(* IEC 61131-3 sources: SIGMATEK-Jumag-Utils-Examples/edgeDetection/Class/Class0, 1 file *)

(* ---- Class0.st ---- *)
(*!
<Class
	Name               = "Class0"
	Revision           = "0.0"
	RealtimeTask       = "false"
	CyclicTask         = "true"
	DefCyclictime      = "100 ms"
	BackgroundTask     = "false"
	Sigmatek           = "false"
	OSInterface        = "false"
	HighPriority       = "false"
	Automatic          = "false"
	UpdateMode         = "Prescan"
	SharedCommandTable = "true"
	Objectsize         = "(660,120)">
	<Channels>
		<Server Name="ClassSvr" Visualized="false" Initialize="false" WriteProtected="true" Retentive="false"/>
		<Server Name="fallingTriggered" Visualized="false" Initialize="false" WriteProtected="false" Retentive="false"/>
		<Server Name="risingTriggered" Visualized="false" Initialize="false" WriteProtected="false" Retentive="false"/>
		<Server Name="targetValue" Visualized="false" Initialize="true" WriteProtected="false" Retentive="false"/>
		<Client Name="signal" Required="true" Internal="false"/>
	</Channels>
	<Dependencies>
		<Files>
			<File Path=".\Source\edgeDetection.c"/>
		</Files>
	</Dependencies>
</Class>
*)
Class0 : CLASS
  //Servers:
	ClassSvr 	: SvrChCmd_DINT;
	targetValue 	: SvrCh_DINT;
	risingTriggered 	: SvrCh_DINT;
	fallingTriggered 	: SvrCh_DINT;
  //Clients:
	signal 	: CltCh_DINT;
  //Variables:
		oldSignal0 	: DINT;
		oldSignal1 	: DINT;
  //Functions:

	FUNCTION VIRTUAL GLOBAL CyWork
		VAR_INPUT
			EAX 	: UDINT;
		END_VAR
		VAR_OUTPUT
			state (EAX) 	: UDINT;
		END_VAR;
  //Tables:
	FUNCTION @STD
		VAR_OUTPUT
			ret_code	: CONFSTATES;
		END_VAR;
	FUNCTION GLOBAL TAB @CT_;
END_CLASS;

Function Global __cdecl rTrig_DINT
VAR_INPUT
  INPUT : DINT;
  PREV : ^DINT;
  TRIGGER : DINT;
END_VAR
VAR_OUTPUT
  Q : BOOL;
END_VAR;

Function Global __cdecl fTrig_DINT
VAR_INPUT
  INPUT : DINT;
  PREV : ^DINT;
  TRIGGER : DINT;
END_VAR
VAR_OUTPUT
  Q : BOOL;
END_VAR;

FUNCTION VIRTUAL GLOBAL Class0::CyWork
	VAR_INPUT
		EAX 	: UDINT;
	END_VAR
	VAR_OUTPUT
		state (EAX) 	: UDINT;
	END_VAR

  signal := signal.Read();

  risingTriggered := rTrig_DINT(INPUT:= signal, PREV:= #oldSignal0, TRIGGER:= targetValue);

  fallingTriggered := fTrig_DINT(INPUT:= signal, PREV:= #oldSignal1, TRIGGER:= targetValue);

	state := READY;

END_FUNCTION
